TYPE ST_CycleTest :
STRUCT
	//enter cycle test mode
	m_enterCycleTestMode:ARRAY[1..g_sArmNum] OF BOOL;

	//enter cycle test mode
	m_enterCycleTestModeSetup:ARRAY[1..g_sArmNum] OF BOOL;

	//enter car cycle mode
	m_carEnterCycleTest:BOOL;

	//target joint position
	m_targetJntPos:ARRAY[1..g_sArmNum,1..2] OF Vec8d := [[-37.0,-30,510.0,5(0)], [70,-105,280.0,5(360)],
																								[-55.0,-30,510.0,5(0)], [30,-105,280.0,5(360)],
																								[40,-27,510.0,5(0)], [-40,-107,280.0,5(360)],
																								[40,-27,510.0,5(0)], [-40,-107,280.0,5(360)]];
	
	m_targetJntPosSetup:ARRAY[1..g_sArmNum,1..2] OF Vec5d := [[2(0), 70, 160, 60], [2(0), 100, 155, 50],
																											[2(0), 70, 120, 60], [2(0), 100.18, 115, 50],
																											[2(0), 70, 72, 60], [2(0), 100, 80, 50],
																											[2(0), 70, 10, 60], [2(0), 100, 0, 50]];
;
	m_targetJntPosCar:ARRAY[1..2] OF Vec8d := [[4(0),50.0, -20, 50, -60],     [2(-33), 2(0), 650.0, 20.0,  450.0, 60.0]];
	
	//cycle number and motion point number
	m_targetCycleNum:ARRAY[1..g_sArmNum] OF INT := [4(200)];
	m_curCycleNum:ARRAY[1..g_sArmNum] OF INT;
	m_curPointNum:ARRAY[1..g_sArmNum] OF INT;
	
	//cycle time
	m_tgtCycleTime:ARRAY[1..g_sArmNum] OF LREAL; //hour
	m_curCycleTime:ARRAY[1..g_sArmNum] OF LREAL; //hour
	m_curCycleTimeCar:LREAL;
	
	//cycle number and motion point number of car
	m_targetCycleNumCar:INT;
	m_curCycleNumCar:INT;
	m_curPointNumCar:INT;
	
	m_disableSlaveJntMotion:ARRAY[1..g_sArmNum] OF Vec8b := [4([8(FALSE)])];
	m_disableSetupJntMotion:ARRAY[1..g_sArmNum] OF Vec5b := [4([3(TRUE),2(FALSE)])];
	m_disableCartJntMotion : Vec8b := [4(TRUE),4(FALSE)];
	
	//target joint velocity
	m_targetJntVelSlave :ARRAY [1..g_sArmNum] OF Vec8d := [4([30.0, 30.0, 30.0, 5(180)])];
	m_targetJntVelSetup :ARRAY [1..g_sArmNum] OF Vec5d := [4([2(0),5.0, 30.0, 30.0])];
	m_targetJntVelCar:Vec8d :=[4(0.0), 30.0, 5.0, 30.0, 5.0];
	
	
	
	m_carEnterESDTest:BOOL;
	m_enterESDTestSetup:ARRAY[1..g_sArmNum] OF BOOL;
	m_enterESDTest:ARRAY[1..g_sArmNum] OF BOOL;
	
	//start motion flag
	m_startMotion:ARRAY[1..g_sArmNum] OF BOOL;
	
	//start motion flag
	m_startMotionSetup:ARRAY[1..g_sArmNum] OF BOOL;
	m_startMotionCar:BOOL;
		
	//slave arm motor encoder and joint encoder
	m_slaveArmMotorEncoder:ARRAY[1..g_sArmNum] OF Vec8di;
	m_slaveArmjntEncoder:ARRAY[1..g_sArmNum] OF Vec8di;
	
	//setup arm motor encoder and joint encoder
	m_setupArmMotorEncoder:ARRAY[1..g_sArmNum] OF Vec5di;
	m_setupArmjntEncoder:ARRAY[1..g_sArmNum] OF Vec5di;
	
	//car joint motor encoder and joint encoder
	m_cartMotorEncoder:Vec8di;
	m_cartjntEncoder:Vec8di;
	
	//actual joint position
	m_actJntPos:ARRAY[1..g_sArmNum] OF Vec8d;
	m_actJntPosSetup:ARRAY[1..g_sArmNum] OF Vec5d;
	m_actJntPosCar:Vec8d;
	
	//point sum
	m_pointSum:ARRAY[1..g_sArmNum] OF INT;
	m_pointSumCar:INT;
	
	m_tgtCycleTimeCar:LREAL; //hours
	
	//step number
	m_stepNum:ARRAY[1..g_sArmNum] OF INT;
	m_stepNumSetup:ARRAY[1..g_sArmNum] OF INT;
	m_stepNumCar:INT;
	
	
	//joint enable
	m_jntEnable:ARRAY[1..g_sArmNum] OF Vec8i;
	m_jntEnableSetup:ARRAY[1..g_sArmNum] OF Vec5i;
		
	//motion pause and finish
	m_pause:ARRAY[1..g_sArmNum] OF BOOL;
	m_finish:ARRAY[1..g_sArmNum] OF BOOL;
	m_pauseCar:BOOL;
	m_finishCar:BOOL;
	
	//arrive flag
	m_arrived:ARRAY[1..g_sArmNum] OF BOOL;
	
	//defult target joint velocity
	m_defultTargetJntVel:Vec8d:=[0.5,0.5,0.05,0.5,0.5,0.5,0.5,0.5];
	
	//defult target joint velocity
	m_defultTargetJntVelSetup:Vec5d:=[1,1,0.050,0.5,0.5];
	
	//defult target joint velocity
	m_defultTargetJntVelCar:Vec8d:=[1,1,1,1,  0.050,0.5,0.050,0.5];		
	
		
	//target joint velocity
	m_targetJntVelN8:ARRAY[1..g_sArmNum] OF Vec8d;
	
	//point id for cover command position---car
	m_pntIdForCoverCmdCar:INT;
	
		//cover command position
	m_coverCmdPos:ARRAY[1..g_sArmNum] OF BOOL;
	
	//point id for cover command position
	m_pntIdForCoverCmd:ARRAY[1..g_sArmNum] OF INT;
	
	//cover command position---car
	m_coverCmdPosCar:BOOL;
END_STRUCT
END_TYPE

(* stored: Version 1.1.0.1, ProductVersion 3.1.4024.11
   DUT ST_CycleTest: Id {4d9eb782-72d4-4cf6-b3fc-606540001649} *)
